// TIA Portal V20 export
VAR_GLOBAL   // PLC tag table "LKinCtrl_Constants"
END_VAR
VAR_GLOBAL CONSTANT   // user constants
   LKINCTRL_MC_MOVELINEARREL : Int := 2;   // cmdType for linear relative command
   LKINCTRL_FM_SET_BEFORE_AND_NO_RESET : USInt := 1;   // set flag before cmd and no reset
   LKINCTRL_MC_ACTIVATE_KIN_ZONE : Int := 34;   // cmdType for activating a workspace zone
   LKINCTRL_MC_MOVELINEARABS : Int := 1;   // cmdType for linear absolute command
   LKINCTRL_FM_SET_AFTER_AND_NO_RESET_AND_WAIT_FOR_ACKNOWLEDGE : USInt := 15;   // set flag after cmd and wait for external reset
   LKINCTRL_NO_OF_PATHDATA_PREBUFFER_ELEMENTS : Int := 5;   // number of PreBuffer elements
   LKINCTRL_FM_RESET_BEFORE : USInt := 20;   // reset flag at start of command
   LKINCTRL_FM_NO_SET_AND_WAIT_FOR_FALSE_ONCE : USInt := 25;   // do not set or reset flag but wait for flag to be false once during command
   LKINCTRL_TABLE_MASK_ARRAY_ENTRIES : DInt := 10;   // maximum size of searchable table
   LKINCTRL_CS_USER_FRAME_4 : Int := 14;   // select fourth user frame
   LKINCTRL_MC_MOVEDIRECTREL : Int := 6;   // cmdType for move direct relative command
   LKINCTRL_FM_DEACTIVATED : USInt := 0;   // flag deactiavted
   LKINCTRL_FM_SET_BEFORE_AND_RESET_AFTER_ONE_CYCLE : USInt := 3;   // set flag before cmd and reset after one cycle
   LKINCTRL_MC_SET_USER_FRAME : Int := 21;   // cmdType for set user frame
   LKINCTRL_CS_NO_OF_FIRST_USER_FRAME : Int := 11;   // index of first user frame
   LKINCTRL_CONFIG_END_OFFSET_COMP : Int := 40;   // cmdType for ending offset compensation
   LKINCTRL_CMD_WAIT_TIME : Int := 100;   // cmdType for wait time command
   LKINCTRL_COMP_RIGHT : Int := 2;   // tool radius compensation to the right
   LKINCTRL_MC_DEFINE_KIN_ZONE : Int := 33;   // cmdType for definining workspace zone
   LKINCTRL_MC_DESYNC_CONVEYOR : Int := 50;   // cmdType for conveyor desync
   LKINCTRL_MC_ACTIVATE_TOOL : Int := 23;   // cmdType for activating a tool
   LKINCTRL_MC_MOVECIRCULARABS : Int := 3;   // cmdType for circular absolute command
   LKINCTRL_CS_USER_FRAME_3 : Int := 13;   // select third user frame
   LKINCTRL_NO_OF_SETFLAGS_BUFFER_ELEMENTS : Int := 15;   // set as double of LKINCTRL_NO_OF_PATHDATA_PREBUFFER_ELEMENTS
   LKINCTRL_TABLE_TYPE_NONSELECTABLE : USInt := 2;   // constant for type non selectable table
   LKINCTRL_CS_USER_FRAME_2 : Int := 12;   // select second user frame
   LKINCTRL_CIRCMODE_GCODE : Int := 3;   // circMode used in GCode
   LKINCTRL_FM_SET_BEFORE_AND_NO_RESET_AND_WAIT_FOR_ACKNOWLEDGE : USInt := 5;   // set flag before cmd and wait for external reset
   LKINCTRL_CS_NO_OF_LAST_USER_FRAME : Int := 15;   // index of last user frame
   LKINCTRL_MC_ACTIVATE_WS_ZONE : Int := 31;   // cmdType for activating a workspace zone
   LKINCTRL_CS_USER_FRAME_1 : Int := 11;   // select first user frame
   LKINCTRL_MC_DEACTIVATE_WS_ZONE : Int := 32;   // cmdType for deactivating workspace zone
   LKINCTRL_FM_DISTANCE_TOLERANCE : LReal := 0.01;   // tolerance for flagmode 10
   LKINCTRL_CONFIG_START_OFFSET_COMP_LEFT : Int := 41;   // cmdType for starting offset compensation left
   LKINCTRL_FM_SET_BEFORE_AND_RESET_AFTER : USInt := 2;   // set flag before cmd and reset after
   LKINCTRL_MC_MOVECIRCULARREL : Int := 4;   // cmdType for circular relative command
   LKINCTRL_OUTER_CORNER : Int := 1;   // Outer corner (linear / linear intersection)
   LKINCTRL_INNER_CORNER : Int := 2;   // Inner corner (linear / linear intersection)
   LKINCTRL_FM_NO_SET_AND_WAIT_FOR_TRUE_ONCE : USInt := 26;   // do not set or reset flag but wait for flag to be true once during command
   LKINCTRL_MC_SHIFT_CS_REL : Int := 60;   // cmdType for relative shift of CS
   LKINCTRL_FM_SET_AT_REMAINING_DISTANCE : USInt := 10;   // set flag at remaining distance
   LKINCTRL_MC_DEACTIVATE_KIN_ZONE : Int := 35;   // cmdType for deactivating workspace zone
   LKINCTRL_COMP_LEFT : Int := 1;   // tool radius compensation to the left
   LKINCTRL_FM_SET_AFTER_AND_RESET_AFTER_ONE_CYCLE : USInt := 13;   // set flag after cmd and reset after one cycle
   LKINCTRL_CONFIG_START_OFFSET_COMP_RIGHT : Int := 42;   // cmdType for starting offset compensation right
   LKINCTRL_CS_USER_FRAME_5 : Int := 15;   // select fifth user frame
   LKINCTRL_TABLE_TYPE_SELECTABLE : USInt := 1;   // constant for type regular table
   LKINCTRL_MC_TRACKCONVEYORBELT : Int := 10;   // cmdType for track conveyor belt command
   LKINCTRL_NO_OF_VALID_BITS : Int := 6;   // number of valid bits in PathDataElement_advanced
   LKINCTRL_MC_SET_OCS_FRAME : Int := 20;   // cmdType for set frame command
   LKINCTRL_FM_SET_AFTER_AND_NO_RESET : USInt := 11;   // set flag after cmd and no reset
   LKINCTRL_MC_MOVEDIRECTABS : Int := 5;   // cmdType for move direct absolute command
   LKINCTRL_CMD_FLAG_ONLY : Int := 0;   // cmdType for flagOnly command (no motion)
   LKINCTRL_MC_DEFINE_WS_ZONE : Int := 30;   // cmdType for definining workspace zone
   LKINCTRL_MC_RESET_SHIFT : Int := 61;   // cmdType for resetting relative shift of CS
   LKINCTRL_FM_RESET_AFTER : USInt := 21;   // reset flag at end of command
   LKINCTRL_PI : LReal := 3.1415926535897932846264;   // constant value for pi
   LKINCTRL_FM_RESET_AT_REMAINING_DISTANCE : USInt := 22;   // reset flag if remaining distance of current command is reached
   LKINCTRL_MC_MOVELINEARPICKANDPLACE : Int := 11;   // cmdType for linear pick and place command sequence
   LKINCTRL_MC_SET_TOOL_FRAME : Int := 22;   // cmdType for defining tool frame
   LKINCTRL_DEFAULT_TO_NAME : WString := '- - -';   // Default name for technology objects
   LKINCTRL_KINEMATICS_TCS : DInt := 3;
   LKINCTRL_KINEMATICS_KINEMATICSZONES : DInt := 10;
   LKINCTRL_KINEMATICS_ZONE_STATE_VIOLATED : UInt := 3;   // Zone is valid, active and violated
   LKINCTRL_KINEMATICS_ZONE_STATE_INVALID : UInt := 0;   // Zone is invalid, inactive and not violated
   LKINCTRL_KINEMATICS_ZONE_STATE_VALID : UInt := 1;   // Zone is valid but not inactive and not violated
   LKINCTRL_KINEMATICS_WORKSPACEZONES : DInt := 10;
   LKINCTRL_KINEMATICS_OCS : DInt := 3;
   LKINCTRL_KINEMATICS_ZONE_STATE_ACTIVE : UInt := 2;   // Zone is valid and active but not violated
   LKINCTRL_KINEMATICS_CONVEYOR_TRACKING : UInt := 3;
   LKINCTRL_KINEMATICS_AXES : DInt := 6;
   LKINCTRL_MEAS_CMD_WITH_ACK : USInt := 2;   // continue after measurement command only with acknowledge
   LKINCTRL_MEAS_CMD_WO_ACK : USInt := 1;   // continue after measurement command without acknowledge
   LKINCTRL_DEFAULT_NAME : WString := '- - -';   // default name of points in datatype
   LKINCTRL_DEFAULT_NAME_STRING : String := '- - -';   // default name of strings in datatype
   LKINCTRL_NO_OF_PATHDATA_ELEMENTS_ADVANCED : Int := 200;   // LEGACY / Length of LKinCtrl_typePathData_advanced
   LKINCTRL_NO_OF_PATHDATA_ELEMENTS_REDUCED : Int := 10;   // LEGACY / Length of LKinCtrl_typePathData_reduced
END_VAR
